FUNCTION_BLOCK FB_SmartHeater
VAR 
    bIsOn : BOOL;
    rTemperature   : REAL;
    nStartCounter  : INT;
	rMaxTemperature : REAL := 120.0;
END_VAR

VAR CONSTANT
    sSerialNumber : STRING := 'HTR-2026-001';
END_VAR

PROPERTY SerialNumber : STRING
GET
  SerialNumber := sSerialNumber;
END_GET
SET
END_SET
END_PROPERTY

PROPERTY StartCount : INT
GET
StartCount := nStartCounter;
END_GET
SET
END_SET
END_PROPERTY

PROPERTY Temperature : REAL
GET
Temperature := rTemperature;
END_GET
SET
  IF bIsOn AND Temperature <= rMaxTemperature THEN
        rTemperature := Temperature;
    END_IF
END_SET
END_PROPERTY

METHOD TurnOff : BOOL
VAR_INPUT
END_VAR
bIsOn := FALSE;
END_METHOD

METHOD TurnOn : BOOL
VAR_INPUT
END_VAR
IF NOT bIsOn THEN
    bIsOn := TRUE;
    nStartCounter := nStartCounter + 1;
END_IF
END_METHOD

END_FUNCTION_BLOCK

(* stored: Version 1.1.0.1, ProductVersion 3.1.4024.16
   POU FB_SmartHeater: Id {bcdc58e1-c42d-4e8a-827c-1b223fca30d2}, SpecialFunc None
   Property SerialNumber: Id {86fef662-6a18-4a03-ba6b-fac36230d6f6}
   Get Get: Id {322da664-80c8-4dd7-bf95-0257cb6cf4e2}
   Set Set: Id {13628f6d-ec22-42d4-bfea-1f0aefcddd1e}
   Property StartCount: Id {51a7686f-552e-473a-b753-b62ed7dff70f}
   Get Get: Id {aa1fd66c-1166-4b4b-a377-4a2f7afa6a5a}
   Set Set: Id {8db8b32c-cd82-4f08-a8f0-f49d5712b45b}
   Property Temperature: Id {3f884351-186a-475a-ae48-a9d0e540e80b}
   Get Get: Id {117fff14-e27b-409e-943a-a827336a400e}
   Set Set: Id {b8b2dcd1-0c27-4767-b500-034436f5e8c4}
   Method TurnOff: Id {50e567f8-46d1-4103-993b-eacc744c72af}
   Method TurnOn: Id {58ecfa5c-b239-42d2-9c7e-5f3bc9d882fa} *)
